ABB RAPID module: PLC_Interface.mod

MODULE PLC_Interface
    !***************************************************************************
    ! PLC Interface Module for Robot Communication
    !***************************************************************************
    ! Description: RAPID module for ABB robot to communicate with Siemens PLC
    ! Purpose: Robot-side interface for coordinate exchange system
    ! Version: 1.0
    ! Date: 17/07/2025
    !
    ! This module provides the robot-side interface for communicating with
    ! the Siemens S7-400H PLC via PROFIBUS-DP or Ethernet
    !***************************************************************************

    ! System parameters
    CONST num PLC_UPDATE_RATE := 0.1;      ! Update rate in seconds
    CONST num PLC_TIMEOUT := 5.0;          ! Communication timeout
    CONST num MAX_COORDINATE_SETS := 10;   ! Maximum coordinate sets
    CONST num MAX_AREAS := 2;              ! Maximum areas

    ! PLC communication data types
    RECORD plc_command_data
        num command_word;       ! Command from PLC
        num status_word;        ! Status to PLC
        num area_selection;     ! Area number (1 or 2)
        num coordinate_set;     ! Set number (1-10)
        num x_coordinate;       ! X coordinate in mm
        num y_coordinate;       ! Y coordinate in mm
        num z_coordinate;       ! Z coordinate in mm
        num rx_rotation;        ! RX rotation in degrees*100
        num ry_rotation;        ! RY rotation in degrees*100
        num rz_rotation;        ! RZ rotation in degrees*100
        num gripper_command;    ! Gripper command (0=open, 1=close)
        num speed_override;     ! Speed override (10-100%)
        num motion_type;        ! Motion type (1=linear, 2=joint)
        num precision;          ! Precision mode (1=fine, 2=coarse)
        num timestamp;          ! Timestamp
        num error_code;         ! Error code
    ENDRECORD

    RECORD robot_feedback_data
        num robot_command;      ! Command received
        num robot_status;       ! Current robot status
        num current_area;       ! Current area
        num current_set;        ! Current set
        num current_x;          ! Current X position
        num current_y;          ! Current Y position
        num current_z;          ! Current Z position
        num current_rx;         ! Current RX rotation
        num current_ry;         ! Current RY rotation
        num current_rz;         ! Current RZ rotation
        num motion_status;      ! Motion status
        num gripper_feedback;   ! Gripper feedback
        num current_speed;      ! Current speed
        num path_progress;      ! Path progress percentage
        num execution_time;     ! Execution time in ms
        num robot_error_code;   ! Robot error code
        num feedback_timestamp; ! Feedback timestamp
    ENDRECORD

    ! Global variables
    VAR plc_command_data plc_command;
    VAR robot_feedback_data robot_feedback;
    VAR bool plc_connected := FALSE;
    VAR bool command_pending := FALSE;
    VAR bool motion_active := FALSE;
    VAR bool emergency_stop_active := FALSE;
    VAR num last_command := 0;
    VAR num current_error_code := 0;
    VAR robtarget coordinate_buffer{MAX_AREAS, MAX_COORDINATE_SETS};
    VAR speeddata motion_speed;
    VAR zonedata motion_zone;

    ! Command constants
    CONST num CMD_NO_COMMAND := 0;
    CONST num CMD_WRITE_COORDINATE := 1;
    CONST num CMD_READ_COORDINATE := 2;
    CONST num CMD_EXECUTE_COORDINATE := 3;
    CONST num CMD_GET_POSITION := 4;
    CONST num CMD_STOP_MOTION := 5;
    CONST num CMD_RESET_ERROR := 6;
    CONST num CMD_GET_STATUS := 7;
    CONST num CMD_EMERGENCY_STOP := 8;
    CONST num CMD_CLEAR_ALL := 9;
    CONST num CMD_VALIDATE_COORDINATE := 10;

    ! Status constants
    CONST num STATUS_IDLE := 0;
    CONST num STATUS_COMMAND_RECEIVED := 1;
    CONST num STATUS_PROCESSING := 2;
    CONST num STATUS_COMPLETED := 3;
    CONST num STATUS_ERROR := 4;
    CONST num STATUS_WARNING := 5;
    CONST num STATUS_BUSY := 6;
    CONST num STATUS_ROBOT_NOT_READY := 7;
    CONST num STATUS_COMMUNICATION_ERROR := 8;
    CONST num STATUS_VALIDATION_FAILED := 9;
    CONST num STATUS_TIMEOUT := 10;

    ! Error codes
    CONST num ERR_NO_ERROR := 0;
    CONST num ERR_INVALID_COMMAND := 1;
    CONST num ERR_INVALID_AREA := 2;
    CONST num ERR_INVALID_SET := 3;
    CONST num ERR_COORDINATE_OUT_OF_RANGE := 4;
    CONST num ERR_ROBOT_NOT_READY := 5;
    CONST num ERR_MOTION_ERROR := 6;
    CONST num ERR_COMMUNICATION_ERROR := 7;
    CONST num ERR_SAFETY_ERROR := 8;
    CONST num ERR_GRIPPER_ERROR := 9;
    CONST num ERR_TIMEOUT := 10;

    !***************************************************************************
    ! PROC PLC_Interface_Main
    ! Main procedure for PLC interface
    !***************************************************************************
    PROC PLC_Interface_Main()
        ! Initialize system
        Initialize_PLC_Interface;

        ! Main communication loop
        WHILE TRUE DO
            ! Read command from PLC
            Read_PLC_Command;

            ! Process command
            Process_PLC_Command;

            ! Update robot feedback
            Update_Robot_Feedback;

            ! Send feedback to PLC
            Send_PLC_Feedback;

            ! Wait for next cycle
            WaitTime PLC_UPDATE_RATE;
        ENDWHILE
    ENDPROC

    !***************************************************************************
    ! PROC Initialize_PLC_Interface
    ! Initialize PLC interface system
    !***************************************************************************
    PROC Initialize_PLC_Interface()
        ! Initialize command data
        plc_command.command_word := CMD_NO_COMMAND;
        plc_command.status_word := STATUS_IDLE;
        plc_command.area_selection := 1;
        plc_command.coordinate_set := 1;
        plc_command.x_coordinate := 0;
        plc_command.y_coordinate := 0;
        plc_command.z_coordinate := 300;
        plc_command.rx_rotation := 0;
        plc_command.ry_rotation := 0;
        plc_command.rz_rotation := 0;
        plc_command.gripper_command := 0;
        plc_command.speed_override := 50;
        plc_command.motion_type := 1;
        plc_command.precision := 1;
        plc_command.timestamp := 0;
        plc_command.error_code := ERR_NO_ERROR;

        ! Initialize feedback data
        robot_feedback.robot_command := CMD_NO_COMMAND;
        robot_feedback.robot_status := STATUS_IDLE;
        robot_feedback.current_area := 1;
        robot_feedback.current_set := 1;
        robot_feedback.current_x := 0;
        robot_feedback.current_y := 0;
        robot_feedback.current_z := 0;
        robot_feedback.current_rx := 0;
        robot_feedback.current_ry := 0;
        robot_feedback.current_rz := 0;
        robot_feedback.motion_status := 0;
        robot_feedback.gripper_feedback := 0;
        robot_feedback.current_speed := 0;
        robot_feedback.path_progress := 0;
        robot_feedback.execution_time := 0;
        robot_feedback.robot_error_code := ERR_NO_ERROR;
        robot_feedback.feedback_timestamp := 0;

        ! Initialize coordinate buffer
        Initialize_Coordinate_Buffer;

        ! Initialize motion parameters
        motion_speed := v50;
        motion_zone := fine;

        ! Reset flags
        command_pending := FALSE;
        motion_active := FALSE;
        emergency_stop_active := FALSE;
        last_command := CMD_NO_COMMAND;
        current_error_code := ERR_NO_ERROR;

        ! Set connection status
        plc_connected := TRUE;

        ! Log initialization
        TPWrite "PLC Interface initialized successfully";
    ENDPROC

    !***************************************************************************
    ! PROC Initialize_Coordinate_Buffer
    ! Initialize coordinate buffer with default values
    !***************************************************************************
    PROC Initialize_Coordinate_Buffer()
        VAR num area;
        VAR num set;

        FOR area FROM 1 TO MAX_AREAS DO
            FOR set FROM 1 TO MAX_COORDINATE_SETS DO
                coordinate_buffer{area, set} := [[0, 0, 300], [1, 0, 0, 0], [0, 0, 0, 0], [9E9, 9E9, 9E9, 9E9, 9E9, 9E9]];
            ENDFOR
        ENDFOR
    ENDPROC

    !***************************************************************************
    ! PROC Read_PLC_Command
    ! Read command from PLC via PROFIBUS or Ethernet
    !***************************************************************************
    PROC Read_PLC_Command()
        ! This would be implemented with specific PLC communication instructions
        ! For PROFIBUS-DP: Use DeviceNet or similar instructions
        ! For Ethernet: Use socket communication

        ! Example implementation (would be hardware-specific):
        ! ReadDeviceData "PLC_Device", plc_command;

        ! For simulation purposes, we'll assume the command is already available
        ! In real implementation, replace with actual PLC communication code

        ! Check for communication errors
        IF plc_connected = FALSE THEN
            current_error_code := ERR_COMMUNICATION_ERROR;
            robot_feedback.robot_status := STATUS_COMMUNICATION_ERROR;
            RETURN;
        ENDIF

        ! Validate received command
        IF plc_command.command_word < CMD_NO_COMMAND OR plc_command.command_word > CMD_VALIDATE_COORDINATE THEN
            current_error_code := ERR_INVALID_COMMAND;
            robot_feedback.robot_status := STATUS_ERROR;
            RETURN;
        ENDIF

        ! Check for new command
        IF plc_command.command_word <> last_command AND plc_command.command_word <> CMD_NO_COMMAND THEN
            command_pending := TRUE;
            robot_feedback.robot_status := STATUS_COMMAND_RECEIVED;
            TPWrite "New command received: " + NumToStr(plc_command.command_word, 0);
        ENDIF
    ENDPROC

    !***************************************************************************
    ! PROC Process_PLC_Command
    ! Process received PLC command
    !***************************************************************************
    PROC Process_PLC_Command()
        ! Skip if no command pending
        IF command_pending = FALSE THEN
            RETURN;
        ENDIF

        ! Check emergency stop
        IF emergency_stop_active = TRUE THEN
            robot_feedback.robot_status := STATUS_ERROR;
            robot_feedback.robot_error_code := ERR_SAFETY_ERROR;
            RETURN;
        ENDIF

        ! Set processing status
        robot_feedback.robot_status := STATUS_PROCESSING;

        ! Process command based on type
        TEST plc_command.command_word
            CASE CMD_WRITE_COORDINATE:
                Execute_Write_Coordinate;
            CASE CMD_READ_COORDINATE:
                Execute_Read_Coordinate;
            CASE CMD_EXECUTE_COORDINATE:
                Execute_Coordinate_Motion;
            CASE CMD_GET_POSITION:
                Execute_Get_Position;
            CASE CMD_STOP_MOTION:
                Execute_Stop_Motion;
            CASE CMD_RESET_ERROR:
                Execute_Reset_Error;
            CASE CMD_GET_STATUS:
                Execute_Get_Status;
            CASE CMD_EMERGENCY_STOP:
                Execute_Emergency_Stop;
            CASE CMD_CLEAR_ALL:
                Execute_Clear_All;
            CASE CMD_VALIDATE_COORDINATE:
                Execute_Validate_Coordinate;
            DEFAULT:
                current_error_code := ERR_INVALID_COMMAND;
                robot_feedback.robot_status := STATUS_ERROR;
        ENDTEST

        ! Update last command
        last_command := plc_command.command_word;
        command_pending := FALSE;
    ENDPROC

    !***************************************************************************
    ! PROC Execute_Write_Coordinate
    ! Execute write coordinate command
    !***************************************************************************
    PROC Execute_Write_Coordinate()
        VAR robtarget target;
        VAR bool validation_result;

        ! Validate area and set
        IF plc_command.area_selection < 1 OR plc_command.area_selection > MAX_AREAS THEN
            current_error_code := ERR_INVALID_AREA;
            robot_feedback.robot_status := STATUS_ERROR;
            RETURN;
        ENDIF

        IF plc_command.coordinate_set < 1 OR plc_command.coordinate_set > MAX_COORDINATE_SETS THEN
            current_error_code := ERR_INVALID_SET;
            robot_feedback.robot_status := STATUS_ERROR;
            RETURN;
        ENDIF

        ! Create target from PLC data
        target.trans.x := plc_command.x_coordinate;
        target.trans.y := plc_command.y_coordinate;
        target.trans.z := plc_command.z_coordinate;

        ! Convert rotations from degrees*100 to quaternions
        target.rot := OrientZYX(plc_command.rz_rotation/100, plc_command.ry_rotation/100, plc_command.rx_rotation/100);

        ! Set configuration (tool and work object would be predefined)
        target.robconf := [0, 0, 0, 0];
        target.extax := [9E9, 9E9, 9E9, 9E9, 9E9, 9E9];

        ! Validate coordinate
        validation_result := Validate_Coordinate(target);
        IF validation_result = FALSE THEN
            current_error_code := ERR_COORDINATE_OUT_OF_RANGE;
            robot_feedback.robot_status := STATUS_VALIDATION_FAILED;
            RETURN;
        ENDIF

        ! Store coordinate in buffer
        coordinate_buffer{plc_command.area_selection, plc_command.coordinate_set} := target;

        ! Update feedback
        robot_feedback.current_area := plc_command.area_selection;
        robot_feedback.current_set := plc_command.coordinate_set;
        robot_feedback.robot_status := STATUS_COMPLETED;
        current_error_code := ERR_NO_ERROR;

        TPWrite "Coordinate written to buffer [" + NumToStr(plc_command.area_selection, 0) + "," + NumToStr(plc_command.coordinate_set, 0) + "]";
    ENDPROC

    !***************************************************************************
    ! PROC Execute_Read_Coordinate
    ! Execute read coordinate command
    !***************************************************************************
    PROC Execute_Read_Coordinate()
        VAR robtarget target;
        VAR EulerAngles euler;

        ! Validate area and set
        IF plc_command.area_selection < 1 OR plc_command.area_selection > MAX_AREAS THEN
            current_error_code := ERR_INVALID_AREA;
            robot_feedback.robot_status := STATUS_ERROR;
            RETURN;
        ENDIF

        IF plc_command.coordinate_set < 1 OR plc_command.coordinate_set > MAX_COORDINATE_SETS THEN
            current_error_code := ERR_INVALID_SET;
            robot_feedback.robot_status := STATUS_ERROR;
            RETURN;
        ENDIF

        ! Get coordinate from buffer
        target := coordinate_buffer{plc_command.area_selection, plc_command.coordinate_set};

        ! Convert to PLC format
        robot_feedback.current_x := target.trans.x;
        robot_feedback.current_y := target.trans.y;
        robot_feedback.current_z := target.trans.z;

        ! Convert quaternions to Euler angles
        euler := RotToEuler(target.rot, OrientZYX);
        robot_feedback.current_rx := euler.rx * 100;
        robot_feedback.current_ry := euler.ry * 100;
        robot_feedback.current_rz := euler.rz * 100;

        ! Update feedback
        robot_feedback.current_area := plc_command.area_selection;
        robot_feedback.current_set := plc_command.coordinate_set;
        robot_feedback.robot_status := STATUS_COMPLETED;
        current_error_code := ERR_NO_ERROR;

        TPWrite "Coordinate read from buffer [" + NumToStr(plc_command.area_selection, 0) + "," + NumToStr(plc_command.coordinate_set, 0) + "]";
    ENDPROC

    !***************************************************************************
    ! PROC Execute_Coordinate_Motion
    ! Execute coordinate motion command
    !***************************************************************************
    PROC Execute_Coordinate_Motion()
        VAR robtarget target;
        VAR speeddata speed;
        VAR zonedata zone;
        VAR num start_time;

        ! Validate area and set
        IF plc_command.area_selection < 1 OR plc_command.area_selection > MAX_AREAS THEN
            current_error_code := ERR_INVALID_AREA;
            robot_feedback.robot_status := STATUS_ERROR;
            RETURN;
        ENDIF

        IF plc_command.coordinate_set < 1 OR plc_command.coordinate_set > MAX_COORDINATE_SETS THEN
            current_error_code := ERR_INVALID_SET;
            robot_feedback.robot_status := STATUS_ERROR;
            RETURN;
        ENDIF

        ! Get target from buffer
        target := coordinate_buffer{plc_command.area_selection, plc_command.coordinate_set};

        ! Set motion parameters
        speed := Calculate_Speed(plc_command.speed_override);
        zone := Calculate_Zone(plc_command.precision);

        ! Check robot readiness
        IF robot_feedback.robot_status = STATUS_ERROR THEN
            current_error_code := ERR_ROBOT_NOT_READY;
            robot_feedback.robot_status := STATUS_ROBOT_NOT_READY;
            RETURN;
        ENDIF

        ! Execute motion
        motion_active := TRUE;
        start_time := GetTime();

        ! Handle gripper command before motion
        IF plc_command.gripper_command = 1 THEN
            Execute_Gripper_Close;
        ELSE
            Execute_Gripper_Open;
        ENDIF

        ! Execute motion based on type
        IF plc_command.motion_type = 1 THEN
            ! Linear motion
            MoveL target, speed, zone, Tool0 \WObj:=WObj0;
        ELSE
            ! Joint motion
            MoveJ target, speed, zone, Tool0 \WObj:=WObj0;
        ENDIF

        ! Calculate execution time
        robot_feedback.execution_time := GetTime() - start_time;

        ! Update feedback
        motion_active := FALSE;
        robot_feedback.robot_status := STATUS_COMPLETED;
        robot_feedback.motion_status := 1; ! Motion completed
        robot_feedback.path_progress := 100;
        current_error_code := ERR_NO_ERROR;

        TPWrite "Motion executed successfully to [" + NumToStr(plc_command.area_selection, 0) + "," + NumToStr(plc_command.coordinate_set, 0) + "]";
    ENDPROC

    !***************************************************************************
    ! PROC Execute_Get_Position
    ! Execute get current position command
    !***************************************************************************
    PROC Execute_Get_Position()
        VAR robtarget current_pos;
        VAR EulerAngles euler;

        ! Get current robot position
        current_pos := CRobT(\Tool:=Tool0 \WObj:=WObj0);

        ! Update feedback with current position
        robot_feedback.current_x := current_pos.trans.x;
        robot_feedback.current_y := current_pos.trans.y;
        robot_feedback.current_z := current_pos.trans.z;

        ! Convert quaternions to Euler angles
        euler := RotToEuler(current_pos.rot, OrientZYX);
        robot_feedback.current_rx := euler.rx * 100;
        robot_feedback.current_ry := euler.ry * 100;
        robot_feedback.current_rz := euler.rz * 100;

        ! Update feedback
        robot_feedback.robot_status := STATUS_COMPLETED;
        current_error_code := ERR_NO_ERROR;

        TPWrite "Current position retrieved";
    ENDPROC

    !***************************************************************************
    ! PROC Execute_Stop_Motion
    ! Execute stop motion command
    !***************************************************************************
    PROC Execute_Stop_Motion()
        ! Stop current motion
        StopMove;

        ! Update status
        motion_active := FALSE;
        robot_feedback.motion_status := 2; ! Motion stopped
        robot_feedback.robot_status := STATUS_COMPLETED;
        current_error_code := ERR_NO_ERROR;

        TPWrite "Motion stopped";
    ENDPROC

    !***************************************************************************
    ! PROC Execute_Reset_Error
    ! Execute reset error command
    !***************************************************************************
    PROC Execute_Reset_Error()
        ! Reset error states
        current_error_code := ERR_NO_ERROR;
        robot_feedback.robot_error_code := ERR_NO_ERROR;
        robot_feedback.robot_status := STATUS_IDLE;
        emergency_stop_active := FALSE;

        ! Clear any system errors (if possible)
        ClearPath;

        TPWrite "Error reset completed";
    ENDPROC

    !***************************************************************************
    ! PROC Execute_Get_Status
    ! Execute get status command
    !***************************************************************************
    PROC Execute_Get_Status()
        ! Status is continuously updated in Update_Robot_Feedback
        ! This command just confirms the request
        robot_feedback.robot_status := STATUS_COMPLETED;
        current_error_code := ERR_NO_ERROR;

        TPWrite "Status request completed";
    ENDPROC

    !***************************************************************************
    ! PROC Execute_Emergency_Stop
    ! Execute emergency stop command
    !***************************************************************************
    PROC Execute_Emergency_Stop()
        ! Stop all motion immediately
        StopMove;

        ! Set emergency stop flag
        emergency_stop_active := TRUE;
        motion_active := FALSE;

        ! Update status
        robot_feedback.robot_status := STATUS_ERROR;
        robot_feedback.robot_error_code := ERR_SAFETY_ERROR;
        current_error_code := ERR_SAFETY_ERROR;

        TPWrite "EMERGENCY STOP ACTIVATED";
    ENDPROC

    !***************************************************************************
    ! PROC Execute_Clear_All
    ! Execute clear all command
    !***************************************************************************
    PROC Execute_Clear_All()
        ! Clear coordinate buffer
        Initialize_Coordinate_Buffer;

        ! Reset status
        robot_feedback.robot_status := STATUS_IDLE;
        robot_feedback.current_area := 1;
        robot_feedback.current_set := 1;
        current_error_code := ERR_NO_ERROR;

        TPWrite "All coordinates cleared";
    ENDPROC

    !***************************************************************************
    ! PROC Execute_Validate_Coordinate
    ! Execute validate coordinate command
    !***************************************************************************
    PROC Execute_Validate_Coordinate()
        VAR robtarget target;
        VAR bool validation_result;

        ! Create target from PLC data
        target.trans.x := plc_command.x_coordinate;
        target.trans.y := plc_command.y_coordinate;
        target.trans.z := plc_command.z_coordinate;
        target.rot := OrientZYX(plc_command.rz_rotation/100, plc_command.ry_rotation/100, plc_command.rx_rotation/100);
        target.robconf := [0, 0, 0, 0];
        target.extax := [9E9, 9E9, 9E9, 9E9, 9E9, 9E9];

        ! Validate coordinate
        validation_result := Validate_Coordinate(target);

        IF validation_result = TRUE THEN
            robot_feedback.robot_status := STATUS_COMPLETED;
            current_error_code := ERR_NO_ERROR;
            TPWrite "Coordinate validation passed";
        ELSE
            robot_feedback.robot_status := STATUS_VALIDATION_FAILED;
            current_error_code := ERR_COORDINATE_OUT_OF_RANGE;
            TPWrite "Coordinate validation failed";
        ENDIF
    ENDPROC

    !***************************************************************************
    ! FUNC Validate_Coordinate
    ! Validate coordinate for reachability and safety
    !***************************************************************************
    FUNC bool Validate_Coordinate(robtarget target)
        VAR bool result := TRUE;

        ! Check workspace limits
        IF target.trans.x < -2000 OR target.trans.x > 2000 THEN
            result := FALSE;
        ENDIF

        IF target.trans.y < -2000 OR target.trans.y > 2000 THEN
            result := FALSE;
        ENDIF

        IF target.trans.z < 0 OR target.trans.z > 1000 THEN
            result := FALSE;
        ENDIF

        ! Check reachability (simplified check)
        ! In real implementation, use more sophisticated reachability analysis
        VAR num distance;
        distance := Sqrt(target.trans.x * target.trans.x + target.trans.y * target.trans.y + target.trans.z * target.trans.z);

        IF distance > 1800 THEN ! Approximate maximum reach
            result := FALSE;
        ENDIF

        RETURN result;
    ENDFUNC

    !***************************************************************************
    ! FUNC Calculate_Speed
    ! Calculate speed data from override percentage
    !***************************************************************************
    FUNC speeddata Calculate_Speed(num override)
        VAR speeddata speed;

        ! Base speed is v100 (100mm/s)
        speed.v_tcp := 100 * (override / 100);
        speed.v_ori := 45 * (override / 100);
        speed.v_leax := 5000 * (override / 100);
        speed.v_reax := 1000 * (override / 100);

        ! Ensure minimum speed
        IF speed.v_tcp < 10 THEN
            speed.v_tcp := 10;
        ENDIF

        RETURN speed;
    ENDFUNC

    !***************************************************************************
    ! FUNC Calculate_Zone
    ! Calculate zone data from precision setting
    !***************************************************************************
    FUNC zonedata Calculate_Zone(num precision)
        VAR zonedata zone;

        IF precision = 1 THEN
            zone := fine;
        ELSE
            zone := z10;
        ENDIF

        RETURN zone;
    ENDFUNC

    !***************************************************************************
    ! PROC Execute_Gripper_Open
    ! Open gripper
    !***************************************************************************
    PROC Execute_Gripper_Open()
        ! This would be implemented with specific gripper I/O
        ! Example: SetDO DO_Gripper_Open, 1;
        ! SetDO DO_Gripper_Close, 0;

        robot_feedback.gripper_feedback := 0;
        TPWrite "Gripper opened";
    ENDPROC

    !***************************************************************************
    ! PROC Execute_Gripper_Close
    ! Close gripper
    !***************************************************************************
    PROC Execute_Gripper_Close()
        ! This would be implemented with specific gripper I/O
        ! Example: SetDO DO_Gripper_Close, 1;
        ! SetDO DO_Gripper_Open, 0;

        robot_feedback.gripper_feedback := 1;
        TPWrite "Gripper closed";
    ENDPROC

    !***************************************************************************
    ! PROC Update_Robot_Feedback
    ! Update robot feedback data
    !***************************************************************************
    PROC Update_Robot_Feedback()
        VAR robtarget current_pos;
        VAR EulerAngles euler;
        VAR speeddata current_speed_data;

        ! Get current position
        current_pos := CRobT(\Tool:=Tool0 \WObj:=WObj0);

        ! Update position feedback
        robot_feedback.current_x := current_pos.trans.x;
        robot_feedback.current_y := current_pos.trans.y;
        robot_feedback.current_z := current_pos.trans.z;

        ! Convert quaternions to Euler angles
        euler := RotToEuler(current_pos.rot, OrientZYX);
        robot_feedback.current_rx := euler.rx * 100;
        robot_feedback.current_ry := euler.ry * 100;
        robot_feedback.current_rz := euler.rz * 100;

        ! Update motion status
        IF motion_active THEN
            robot_feedback.motion_status := 1; ! Motion in progress
        ELSE
            robot_feedback.motion_status := 0; ! Motion idle
        ENDIF

        ! Update current speed (approximation)
        current_speed_data := CSpeedOverride();
        robot_feedback.current_speed := current_speed_data.v_tcp;

        ! Update timestamp
        robot_feedback.feedback_timestamp := GetTime();

        ! Update error code
        robot_feedback.robot_error_code := current_error_code;

        ! Copy command to feedback
        robot_feedback.robot_command := plc_command.command_word;
    ENDPROC

    !***************************************************************************
    ! PROC Send_PLC_Feedback
    ! Send feedback to PLC
    !***************************************************************************
    PROC Send_PLC_Feedback()
        ! This would be implemented with specific PLC communication instructions
        ! For PROFIBUS-DP: Use DeviceNet or similar instructions
        ! For Ethernet: Use socket communication

        ! Example implementation (would be hardware-specific):
        ! WriteDeviceData "PLC_Device", robot_feedback;

        ! For simulation purposes, assume feedback is sent
        ! In real implementation, replace with actual PLC communication code

        ! Check communication status
        IF plc_connected = FALSE THEN
            TPWrite "PLC communication lost";
            RETURN;
        ENDIF

        ! Log feedback sending (for debugging)
        ! TPWrite "Feedback sent: Status=" + NumToStr(robot_feedback.robot_status, 0);
    ENDPROC

    !***************************************************************************
    ! PROC PLC_Interface_Stop
    ! Stop PLC interface (called on program stop)
    !***************************************************************************
    PROC PLC_Interface_Stop()
        ! Stop any active motion
        StopMove;

        ! Reset status
        robot_feedback.robot_status := STATUS_IDLE;
        robot_feedback.robot_error_code := ERR_NO_ERROR;
        motion_active := FALSE;
        command_pending := FALSE;

        ! Send final feedback
        Send_PLC_Feedback;

        ! Set disconnected status
        plc_connected := FALSE;

        TPWrite "PLC Interface stopped";
    ENDPROC

ENDMODULE
